FUNCTION Convert_REAL_TO_DWORD : Hresult
VAR_INPUT
	in : REAL;
	out : REFERENCE TO DWORD;
END_VAR
VAR
	converted : DWORD;
END_VAR
VAR CONSTANT
	INCOMPATIBLE : HRESULT := 16#9811070E;
END_VAR

converted := REAL_TO_DWORD(in);

IF (DWORD_TO_REAL(converted) <> in) THEN
	Convert_REAL_TO_DWORD := INCOMPATIBLE;
	RETURN;
END_IF

out := converted;

END_FUNCTION

(* stored: Version 1.1.0.1, ProductVersion 3.1.4024.12
   POU Convert_REAL_TO_DWORD: Id {d934c707-0901-433f-bf99-af498ded5a6a}, SpecialFunc None *)
